// TwinCAT 3 PLC project TcSocketHelper_MultiClientBinary
// ProgramVersion: 3.1.0.5
// libraries:
//   Tc2_Standard, * (Beckhoff Automation GmbH)
//   Tc2_System, * (Beckhoff Automation GmbH)
//   Tc2_TcpIp, * (Beckhoff Automation GmbH)
//   Tc2_Utilities, * (Beckhoff Automation GmbH)
//   Tc3_Module, * (Beckhoff Automation GmbH)
// project tree:
//   Data types/ ST_ApplicationBinaryData.TcDUT, ST_BinaryFrame.TcDUT, ST_BinaryHeader.TcDUT
//   Global Variables/ Global_Variables.TcGVL
//   POUs/ FB_Client.TcPOU, FB_ClientApplication.TcPOU, FB_ClientConnection.TcPOU, MAIN.TcPOU
//   POUs/Helper POUs/ FB_FrameFifo.TcPOU (not stored), FB_LogFifo.TcPOU (not stored), F_ADSLOGHEXDATA.TcPOU
//   / PlcTaskClient.TcTTO
// real-time tasks:
//   TASK PlcTaskClient: cycle T#10ms, priority 20, ADS port 350

CONFIGURATION TcSocketHelper_MultiClientBinary
    RESOURCE PLC ON TwinCAT3
        TASK PlcTaskClient(INTERVAL := T#10ms, PRIORITY := 20);
        PROGRAM MAIN WITH PlcTaskClient : MAIN;
    END_RESOURCE
END_CONFIGURATION

// ---- Data types/ST_ApplicationBinaryData.TcDUT
(* Simple binary user data (8 byte aligned) *)
TYPE ST_ApplicationBinaryData :
STRUCT
	(* Adapt this structure to match your protocol needs *)
	
	dtTimeStamp : DT		:= DT#2008-12-01-00:00;(* 4 byte *)
	nVelo		: UDINT		:= 0;(* 4 byte *)
	fPos		: LREAL		:= 0.0;(* 8 byte *)
	arr	 		: ARRAY[0..19] OF BYTE;(* 20 byte *)

	sMsg		: STRING	:= 'None';(* 81 byte *)
	reserved	: ARRAY[0..2] OF BYTE;(* Alignment data: 3 byte *)

	(* Total user data size = 120 byte *)
END_STRUCT
END_TYPE

// ---- Data types/ST_BinaryFrame.TcDUT
(* Simple binary TCP/IP frame (8 byte aligned) *)
TYPE ST_BinaryFrame :
STRUCT
	head	: ST_BinaryHeader;(* Frame header (16 byte) *)
	data 	: ST_ApplicationBinaryData;(* User data (120 byte) *)

	(* Total frame size = 136 byte *)
END_STRUCT
END_TYPE

// ---- Data types/ST_BinaryHeader.TcDUT
(* Simple binary TCP/IP frame header (8 byte aligned) *)
TYPE ST_BinaryHeader :
STRUCT
	dwStart		: DWORD	:= 16#BECF1234;	(* Start bytes *)
	cbLength	: UDINT(0..PLCPRJ_BUFFER_SIZE) := 0;(* Max. length of attached binary data *)
	nS			: UDINT := 0;(* Send counter *)
	nR			: UDINT	:= 0;(* Receive counter *)
	
	(* Total header data size = 16 byte *)
END_STRUCT
END_TYPE

// ---- Global Variables/Global_Variables.TcGVL
VAR_GLOBAL CONSTANT
	PLCPRJ_BUFFER_SIZE						: UDINT := 1000;(* Max. internal fifo/receiver buffer size *)

	PLCPRJ_CLIENT_SEND_CYCLE_TIME			: TIME := T#1S;
	PLCPRJ_RECEIVE_POLLING_TIME				: TIME := T#100MS;
	PLCPRJ_RECEIVE_TIMEOUT					: TIME := T#50S;

	(* Some project specific error codes *)
	PLCPRJ_ERROR_RECEIVE_TIMEOUT			: UDINT := 16#8101;(* Receive timeout *)
	PLCPRJ_ERROR_SENDFIFO_OVERFLOW			: UDINT := 16#8102;(* Send fifo overflow *)
	PLCPRJ_ERROR_RECFIFO_OVERFLOW			: UDINT := 16#8103;(* Receive fifo overflow *)
	PLCPRJ_ERROR_INVALID_FRAME_FORMAT		: UDINT := 16#8104;(* Invalid frame format/data *)
END_VAR

// ---- POUs/MAIN.TcPOU
PROGRAM MAIN
VAR
	sSrvNetID			: T_AmsNetID	:= '';(* TwinCAT TCP/IP server network address *)
	bEnable1			: BOOL 			:= TRUE;(* TRUE => Enable client 1 data exchange, FALSE => Disable *)
	bEnable2			: BOOL 			:= FALSE;(* TRUE => Enable client 2 data exchange, FALSE => Disable *)
	bEnable3			: BOOL 			:= FALSE;(* TRUE => Enable client 3 data exchange, FALSE => Disable *)
	bEnable4			: BOOL 			:= FALSE;(* TRUE => Enable client 4 data exchange, FALSE => Disable *)
	bEnable5			: BOOL 			:= FALSE;(* TRUE => Enable client 5 data exchange, FALSE => Disable *)
	bLog				: BOOL			:= TRUE;(* TRUE => Enable log message output, FALSE => Disable *)

	fbClient1	: FB_Client := ( sRemoteHost:= '127.0.0.1',(* Server IP network address *) 
								nRemotePort:= 200,(* Server port number *)
								sPrefix := 'CLIENT1::' );(* Client (connection) instance *)
	fbClient2	: FB_Client := ( sRemoteHost:= '127.0.0.1', nRemotePort:= 200, sPrefix := 'CLIENT2::' );(* Client (connection) instance *)
	fbClient3	: FB_Client := ( sRemoteHost:= '127.0.0.1', nRemotePort:= 200, sPrefix := 'CLIENT3::' );(* Client (connection) instance *)
	fbClient4	: FB_Client := ( sRemoteHost:= '127.0.0.1', nRemotePort:= 200, sPrefix := 'CLIENT4::' );(* Client (connection) instance *)
	fbClient5	: FB_Client := ( sRemoteHost:= '127.0.0.1', nRemotePort:= 200, sPrefix := 'CLIENT5::' );(* Client (connection) instance *)

	fbCloseAll	: FB_SocketCloseAll;
	bInitialize	: BOOL := TRUE;
END_VAR

(* On PLC reset or program download close all old (opened) connections *)
fbCloseAll( sSrvNetID := sSrvNetID, bExecute:= bInitialize );
IF fbCloseAll.bBusy OR fbCloseAll.bError THEN
	RETURN;
END_IF
bInitialize := FALSE;

fbClient1( sSrvNetID := sSrvNetID, bEnable := bEnable1, bLog := bLog );
fbClient2( sSrvNetID := sSrvNetID, bEnable := bEnable2, bLog := bLog );
fbClient3( sSrvNetID := sSrvNetID, bEnable := bEnable3, bLog := bLog );
fbClient4( sSrvNetID := sSrvNetID, bEnable := bEnable4, bLog := bLog );
fbClient5( sSrvNetID := sSrvNetID, bEnable := bEnable5, bLog := bLog );

END_PROGRAM

// ---- POUs/FB_Client.TcPOU
FUNCTION_BLOCK FB_Client
VAR_INPUT
	sSrvNetID	: T_AmsNetID	:= '';(* TwinCAT TCP/IP server network address *)
	sRemoteHost	: T_IPv4Addr 	:= '127.0.0.1';(* Server IP network address *)
	nRemotePort	: UDINT 		:= 200;(* Server port number *)
	bEnable		: BOOL 			:= FALSE;(* TRUE => enable client data exchange, FALSE => disable *)
	bLog		: BOOL 			:= FALSE;(* TRUE => Enable log message output, FALSE => Disable *)
	sPrefix		: STRING 		:= 'CLIENT::';(* Log message description string (allows the identification of log message source) *)
END_VAR
VAR_OUTPUT
	eState		: E_SocketConnectionState := eSOCKET_DISCONNECTED;(* TCP/IP connection state *)
END_VAR
VAR
	fbApplication 	: FB_ClientApplication;(* Client application control function block *)
	fbConnection	: FB_ClientConnection;(* Client data exchange control function block *)
	fbTx 			: FB_FrameFifo;(* Tx fifo *)
	fbRx 			: FB_FrameFifo;(* Rx fifo *)
	fbLog			: FB_LogFifo;(* Log/debug/error fifo *)
END_VAR

(*-------------------------- Trigger data exchange -----------------------------------------------*)
fbConnection( 	sSrvNetID := sSrvNetID, fbRx := fbRx, fbTx := fbTx, fbLog := fbLog, 
				bEnable := bEnable, sRemoteHost := sRemoteHost, nRemotePort := nRemotePort,  
				bLog := bLog, sPrefix := sPrefix, eState=>eState );
	
IF fbConnection.eState = eSOCKET_CONNECTED THEN(* Connection established *)
	fbApplication( fbTx := fbTx, fbRx := fbRx, fbLog := fbLog );
END_IF

END_FUNCTION_BLOCK

// ---- POUs/FB_ClientApplication.TcPOU
(* Sample client application. Adapt this code to match your needs. *)
FUNCTION_BLOCK FB_ClientApplication
VAR_IN_OUT
	fbTx 			: FB_FrameFifo;(* TX fifo *)
	fbRx 			: FB_FrameFifo;(* RX fifo *)
	fbLog			: FB_LogFifo;(* Log message fifo *)
END_VAR
VAR
	stToServer		: ST_ApplicationBinaryData; (* Tx user data *)
	stFromServer	: ST_ApplicationBinaryData; (* Rx user data *)
	sLogMessage 	: T_MaxString := '';(* Log/debug/error message *)

	fbClock			: FB_LocalSystemTime := ( bEnable := TRUE );(* OS clock *)
	fbSndTimer		: TON;(* Cyclic (send) timer *)
END_VAR

(* Refresh clock time *)
fbClock();
IF NOT fbClock.bValid THEN
	RETURN;
END_IF

(*--------------------- Send tx data ------------------------------------------- *)
fbSndTimer( IN := TRUE, PT := PLCPRJ_CLIENT_SEND_CYCLE_TIME );
IF fbSndTimer.Q THEN
	fbSndTimer( IN := FALSE );

	(* Simulate user data *)
	stToServer.dtTimeStamp 	:= SYSTEMTIME_TO_DT( fbClock.systemTime );
	stToServer.fPos 		:= stToServer.fPos + 0.1;
	stToServer.nVelo 		:= stToServer.nVelo + 1;
	stToServer.sMsg 		:= 'Hello world from client!';
	stToServer.arr[0] 		:= stToServer.arr[0] + 1;

	fbTx.AddTail( stPut := stToServer );(* Put user data to the tx fifo *)
	IF NOT fbTx.bOk THEN(* Fifo overflow => Log error *)
		fbLog.Error( sMessage := 'FB_FrameFifo(sender)', nErrID := PLCPRJ_ERROR_SENDFIFO_OVERFLOW );
	END_IF
END_IF

(*------------------------ Fetch rx data -------------------------------------- *)
REPEAT
	fbRx.RemoveHead( );(* fetch data from rx fifo *)
	IF fbRx.bOk THEN(* success *)

		(* TODO: Implement receive handler *)
		stFromServer := fbRx.stGet; 

	END_IF
UNTIL NOT fbRx.bOk
END_REPEAT

(*---------------------- Get log/error messages from log fifo ------------------*)
REPEAT
	fbLog.Remove( );
	IF fbLog.bOk THEN

		(* TODO: Implement log message handler *)
		sLogMessage := fbLog.sGet;

	END_IF
UNTIL NOT fbLog.bOk
END_REPEAT

END_FUNCTION_BLOCK

// ---- POUs/FB_ClientConnection.TcPOU
(* 	This function block implements simple TCP/IP client protocol. *)
FUNCTION_BLOCK FB_ClientConnection
VAR_IN_OUT
	fbTx 		: FB_FrameFifo;(* TX fifo *)
	fbRx 		: FB_FrameFifo;(* RX fifo *)
	fbLog		: FB_LogFifo;(* Log message fifo *)
END_VAR
VAR_INPUT
	sSrvNetID	: T_AmsNetID	:= '';(* TwinCAT TCP/IP server network address *)
	sRemoteHost	: T_IPv4Addr 	:= '127.0.0.1';(* IP address of remote server *)
	nRemotePort	: UDINT			:= 200;(* Remote server port *)
	bEnable		: BOOL			:= FALSE;(* TRUE => Enable/connect, FALSE => Disable/disconnect *)
	tReconnect	: TIME 			:= T#45S;(* Try to reconnect after this time *)
	bLog		: BOOL 			:= FALSE; (* TRUE => Enable debug output, FALSE => Disable debug output *)
	sPrefix		: STRING 		:= 'CLIENT::';(* Log message description string (allows the identification of log message source) *)
END_VAR
VAR_OUTPUT
	eState		: E_SocketConnectionState := eSOCKET_DISCONNECTED;(* TCP/IP connection state *)
END_VAR
VAR
	fbConnect 	: FB_ClientServerConnection;(* Create/release TCP/IP connection *)
	fbSend		: FB_SocketSend;(* Send TCP/IP data *)
	fbReceive	: FB_SocketReceive;(* Receive TCP/IP data *)
	nState 		: BYTE;(* Global state *)
	bSndBusy 	: BOOL;(* Tx state *)
	bRcvBusy 	: BOOL;(* Rx state *)
	bDisconnect	: BOOL;(* Disconnect flag, if set the socket will be closed *)

	fbPollTimer	: TON;(* Rx data poll timer *)
	fbResponseTimer	: TON;(* Response timeout timer *)
	fbReconnectTimer : TON;(* Reconnect timer *)

	nS			: UDINT;(* Send frame counter *)
	nR			: UDINT;(* Received frame counter *)
	cbReceived	: UDINT;(* Count of received data bytes *)
	rxBuffer	: ARRAY[0..PLCPRJ_BUFFER_SIZE] OF BYTE;
	cbFrame		: UDINT;(* Rx frame byte size *)
	stTxFrame	: ST_BinaryFrame;(* Tx frame buffer (inclusive header) *)
	stRxFrame	: ST_BinaryFrame;(* Rx frame buffer (inclusive header) *)
	bAbort		: BOOL;(* Flag to abort frame parsing loop *)
END_VAR

CASE nState OF
	0:(* Create TCP/IP connection *)
		fbConnect( 	sSrvNetID 		:= sSrvNetID,
					nMode			:= SEL( bLog, 0, CONNECT_MODE_ENABLEDBG ),(* Enable/disable debug output *)
					sRemoteHost 	:= sRemoteHost,
					nRemotePort 	:= nRemotePort,
					tReconnect		:= tReconnect,
					bEnable			:= bEnable,
					eState			=> eState );
		IF NOT fbConnect.bBusy THEN
			IF NOT fbConnect.bError THEN
				IF eState = eSOCKET_CONNECTED THEN(* we are connected *)
					
					fbTx.Clear( sPrefix := CONCAT( sPrefix, 'FB_FrameFifo(sender)::' ), bLog := bLog );(* Clear TX fifo (optional) *)
					fbRx.Clear( sPrefix := CONCAT( sPrefix, 'FB_FrameFifo(receiver)::' ), bLog := bLog );(* Clear RX fifo (optional) *)
					fbLog.Clear( sPrefix := sPrefix, bLog := bLog );(* Clear log fifo (optional) *)
					bSndBusy := FALSE;
					bRcvBusy := FALSE;
					bDisconnect := FALSE;
					cbReceived 	:= 0;(* Reset number of received data bytes *)
					nR 			:= 0;(* Reset receive frame counter *)
					nS 			:= 0;(* Reset send frame counter *)

					fbPollTimer( IN := FALSE, PT := T#0S );
					fbResponseTimer( IN := FALSE, PT := PLCPRJ_RECEIVE_TIMEOUT );
					fbReconnectTimer( IN := FALSE, PT := tReconnect );
					
				
					fbLog.Message( sMessage := 'Connection established!', hSocket := fbConnect.hSocket );
					nState 	:= 1;
				END_IF
			ELSE(* Connect error => log error *)
				fbLog.Error( sMessage := 'FB_ClientServerConnection()', nErrID := fbConnect.nErrId );
			END_IF
		END_IF


	1:(* Data exchange state *)
		bDisconnect := NOT bEnable OR bDisconnect;(* User/internal disconnect requested? *)
		IF bDisconnect AND NOT bSndBusy AND NOT bRcvBusy THEN
			bDisconnect := FALSE;
			fbLog.Message( sMessage := 'Closing connection!', hSocket := fbConnect.hSocket );
			nState := 2;(* Disconnect *)
		ELSE

			(* --------------------------- Send tx data --------------------------------- *)
			IF NOT bDisconnect AND NOT bSndBusy THEN
				fbTx.RemoveHead();(* Remove oldest user data entry *)
				IF fbTx.bOk THEN(* Success *)
						
					stTxFrame.data := fbTx.stGet;
					
					(* Append/create some protocol header *)
					stTxFrame.head.dwStart 	:= 16#BECF1234;(* Frame start bytes *)
					stTxFrame.head.cbLength := SIZEOF( stTxFrame.data);(* Set length of user data *)
					stTxFrame.head.nS 		:= nS;(* Number of send frames *)
					stTxFrame.head.nR 		:= nR;(* Number of received frames *)
					
					(* Send frame *)
					fbSend( bExecute := FALSE );
					fbSend(	sSrvNetID 	:= sSrvNetID,
							hSocket		:= fbConnect.hSocket,
							cbLen		:= SIZEOF(stTxFrame),(* Size of header + size of user data *)
							pSrc		:= ADR(stTxFrame),(* Pointer to the frame data *)
							bExecute	:= TRUE );
					bSndBusy := TRUE;
				END_IF
			ELSE(* Wait until send not busy *)
				fbSend( bExecute := FALSE );
				IF NOT fbSend.bBusy THEN
					bSndBusy := FALSE;
					IF NOT fbSend.bError THEN(* No error *)
						nS := nS + 1;(* Increment the number of send frames *)
					ELSE(* Send error => Log error and disconnect *)
						fbLog.Error( sMessage := 'FB_SocketSend()', nErrID := fbSend.nErrId );
						bDisconnect := TRUE;(* Set flag *)
					END_IF
				END_IF
			END_IF
			(* -------------------------------------------------------------------------- *)

			(* ------------------ Get/fetch rx data ------------------------------------- *)
			IF NOT bDisconnect AND NOT bRcvBusy THEN
				fbPollTimer( IN := TRUE );
				IF fbPollTimer.Q THEN
					IF fbRx.cbFree >= SIZEOF(stRxFrame.data) THEN(* Check free rx fifo space *)
						fbPollTimer( IN := FALSE, PT := PLCPRJ_RECEIVE_POLLING_TIME );
						fbReceive( bExecute := FALSE );
						fbReceive( 	sSrvNetId	:= sSrvNetID,
									hSocket		:= fbConnect.hSocket,
									cbLen		:= SIZEOF(rxBuffer) - cbReceived,
									pDest		:= ADR(rxBuffer) + cbReceived,
									bExecute	:= TRUE );
						bRcvBusy := TRUE;
					END_IF
				END_IF
				
			ELSE(* Wait until receive not busy *)
				
				fbReceive( bExecute := FALSE );
				IF NOT fbReceive.bBusy THEN
					bRcvBusy := FALSE;
					IF NOT fbReceive.bError THEN
						IF fbReceive.nRecBytes > 0 THEN (* Some bytes received *)

							fbPollTimer( IN := FALSE, PT := T#0S );(* Bytes received => increase the read (polling) speed *)
							fbResponseTimer( IN := FALSE );(* Bytes received => disable timeout check *)
							cbReceived := cbReceived + fbReceive.nRecBytes;

							(* Parse received bytes *)
							REPEAT
								bAbort := TRUE;(* Set flag *)
								
								IF cbReceived >= SIZEOF(stRxFrame.head) THEN (* All header bytes received => check header data *)
									
									MEMCPY( ADR( stRxFrame.head ), ADR( rxBuffer ), SIZEOF( stRxFrame.head ) );(* Get header data *)
								
									IF (stRxFrame.head.dwStart = 16#BECF1234) (* Check start bytes *)
									AND (stRxFrame.head.nS = nR )(* Check counter (send counter == expected receive counter?) *)
									AND (stRxFrame.head.cbLength <= SIZEOF(stRxFrame.data))(* Check frame (user data) length *)
									THEN
									
										cbFrame := SIZEOF(stRxFrame.head) + stRxFrame.head.cbLength;(* Calculate the expected receive frame length *)
										IF cbReceived >= cbFrame  THEN (* All frame (user data) bytes received? *)
	
											MEMCPY( ADR( stRxFrame ), ADR( rxBuffer ), MIN( SIZEOF(stRxFrame), cbFrame ) );
											fbRx.AddTail( stPut := stRxFrame.data );(* Add user data to the rx fifo *)
											IF fbRx.bOk THEN
												nR := nR + 1;(* Increment receive counter *)

												MEMMOVE( ADR( rxBuffer ), ADR( rxBuffer ) + cbFrame, cbReceived - cbFrame );(* Shift the remaining rx bytes *)
												cbReceived := cbReceived - cbFrame;(* Recalculate the size of the remaining rx bytes *)

												IF fbRx.cbFree >= SIZEOF(stRxFrame.data) THEN
													bAbort := FALSE;(* reset flag, try to parse next frame *)
												END_IF
											ELSE (* Fifo overflow => log error and disconnect *)
												fbLog.Error( sMessage := 'FB_FrameFifo(receiver)', nErrID := PLCPRJ_ERROR_RECFIFO_OVERFLOW );
												bDisconnect := TRUE;(* Set flag *)
												RETURN;
											END_IF

(*										ELSE repeat reading *)
										END_IF

									ELSE(* Receive error => Invalid frame format/data *)
										fbLog.Error( sMessage := 'FB_ClientConnection()', nErrID := PLCPRJ_ERROR_INVALID_FRAME_FORMAT );
										bDisconnect := TRUE;(* Set flag *)
										RETURN;
									END_IF

(*								ELSE repeat reading *)
								END_IF (* IF cbReceived >= SIZEOF(stRxFrame.head) THEN *)

							UNTIL bAbort
							END_REPEAT

						ELSE(* No bytes received *)
							fbResponseTimer( IN := TRUE );(* No bytes received => enable timeout check *)
							IF fbResponseTimer.Q THEN (* Timeout error*)
								fbResponseTimer( IN := FALSE );
								fbLog.Error( sMessage := 'FB_ClientConnection()', nErrID := PLCPRJ_ERROR_RECEIVE_TIMEOUT );
								bDisconnect := TRUE;(* Set flag *)
							END_IF							
						END_IF(* IF fbReceive.nRecBytes > 0 THEN *)

					ELSE(* Receive error => Log error and disconnect *)
						fbLog.Error( sMessage := 'FB_SocketReceive()', nErrID := fbReceive.nErrId );
						bDisconnect := TRUE;(* set flag *)
					END_IF

				END_IF(* IF NOT fbReceive.bBusy THEN *)
				
			END_IF(* IF NOT bDisconnect AND NOT bRcvBusy THEN *)
			(* -------------------------------------------------------------------------- *)
			
			
		END_IF(* IF bDisconnect AND NOT bSndBusy AND NOT bRcvBusy THEN *)


	2:(* Disconnect *)
		fbConnect( bEnable:= FALSE, eState=>eState );
		IF eState = eSOCKET_DISCONNECTED THEN
			fbReconnectTimer( IN := TRUE );(* Please wait some seconds and then try to connect again *)
			IF fbReconnectTimer.Q THEN
				fbReconnectTimer( IN := FALSE );
				nState := 0;
			END_IF
		END_IF


END_CASE

END_FUNCTION_BLOCK

// ---- POUs/Helper POUs/F_ADSLOGHEXDATA.TcPOU
(* This function logs hexadecimal data to the TwinCAT XAE->Error list window *)
FUNCTION F_ADSLOGHEXDATA : DINT
VAR_INPUT
	sPrefix		: STRING;(* Debug message prefix string (allows the identification of log message source) *)
	pBuffer		: PVOID;(* Address of source buffer *)
	cbBuffer	: UDINT;(* Byte size of source buffer *)
END_VAR
VAR
	fbSplit	: FB_MemBufferSplit;
	sArg	: T_MaxString;
	sFormat : STRING;
END_VAR

IF pBuffer = 0 OR cbBuffer = 0 THEN
	RETURN;
END_IF

sFormat := CONCAT( sPrefix, '%s' );
fbSplit.eCmd := eEnumCmd_First;

REPEAT
	fbSplit( pBuffer := pBuffer, cbBuffer := cbBuffer, cbSize := 32 );(* Split binary data to 32 byte segments *)
	IF fbSplit.bOk THEN

		sArg := DATA_TO_HEXSTR( pData := fbSplit.pSegment, cbData := fbSplit.cbSegment, FALSE );(* Convert binary data to hex string *)

		F_ADSLOGHEXDATA := ADSLOGSTR( ADSLOG_MSGTYPE_HINT OR ADSLOG_MSGTYPE_LOG, sFormat, sArg );(* Log hex string *)

		sFormat := '%s';
		fbSplit.eCmd := eEnumCmd_Next;
	END_IF
UNTIL NOT fbSplit.bOk
END_REPEAT

END_FUNCTION
